PROGRAM MAIN
VAR
END_VAR

END_PROGRAM

(* stored: Version 1.1.0.1
   POU MAIN: Id {10618c21-1547-4e83-a456-0820e6a78bd8} *)
